// TIA Portal V20 export
TYPE "typeSequenceControlNodeHomeCheck_topTapeAttachment"
// stored: Namespace Unit1.Em3
   STRUCT
      tapeGetReq { ExternalWritable := 'False'} : Bool;
      tapeGet { ExternalWritable := 'False'} : Bool;
   END_STRUCT;
END_TYPE
